// SIMATIC STEP 7 (V5.x) project hhh_v1_bisai_7_20_20_40
// CPU: CPU 412-3 H
// station: Hardware
// station: SIMATIC 400(1)
// station: P_ADR_BUS
// station: Configuration
// station: PCStation
// station: P_ADR_BUS
// program: S7 Program(1)

SYMBOL_TABLE
"OP_A_LIM"	FB 46	FB 46	// Analog value operating (limited)
"CTRL_PID"	FB 61	FB 61	// PID Control
"MEAS_MON"	FB 65	FB 65	// Meas.value monitoring block
"CONEC"	FB 88	FB 88	// Connection Function Block
"PS"	FB 89	FB 89	// Power Supply Function Block
"OB_BEGIN"	FB 100	FB 100	// CPU Function Block
"SUBNET"	FB 106	FB 106	// SUBNET Function Block
"RACK"	FB 107	FB 107	// RACK Function Block
"OB_DIAG1"	FB 118	FB 118	// OB Diagnostic Function
"CPU_RT"	FB 128	FB 128	// CPU Performance Block
"@SFC_BZL"	FB 245	FB 245	// SFC-State Logic
"@SFC_ESM"	FB 246	FB 246	// SFC-Extended State Management
"@SFC_RTS"	FB 300	FB 300	// SFC-Run-Time System V6
"SUB_R"	FC 62	FC 62	// REAL-Subtraction
"@SFC_INDCALL"	FC 250	FC 250	// SFC-Indirect-Call Function
"ADD4_P"	FC 256	FC 256	// Adder with 4 inputs
"ChkREAL"	FC 260	FC 260	// Check infinite values
"MUL4_P"	FC 262	FC 262	// Multiplier with 4 inputs
"CH_AI"	FC 275	FC 275	// Analog Input
"CH_AO"	FC 276	FC 276	// Analog Output
"PO_UPDAT"	FC 279	FC 279	// Update Process Output
"OB_END"	FC 280	FC 280	// Terminate OB Function Block
"FI1106"	IW 512	WORD	// 产品D混合物料流量
"FI1101"	IW 514	WORD	// 原料A流量
"FI1102"	IW 516	WORD	// 原料B流量
"FI1103"	IW 518	WORD	// 原料混合进料流量
"FI1104"	IW 520	WORD	// 催化剂C流量
"FI1105"	IW 522	WORD	// 反应生成液流量
"FI1107"	IW 524	WORD	//  闪蒸罐顶部循环原料A流量
"FI1201"	IW 526	WORD	// 反应器R101夹套循环上水流量
"FI1202"	IW 528	WORD	//  反应器R101夹套循环回水至预热器流量
"FI1203"	IW 530	WORD	//  反应器R101夹套循环回水至界区流量
"LI1101"	IW 532	WORD	//  混合罐V101液位
"LI1102"	IW 534	WORD	//  反应器R101液位
"LI1201"	IW 536	WORD	//  闪蒸罐V102液位
"TI1101"	IW 538	WORD	//  混合罐V101温度
"TI1102"	IW 540	WORD	//  原料混合进料出预热器E101温度
"TI1103"	IW 542	WORD	//  反应器R101温度
"TI1104"	IW 544	WORD	// 闪蒸罐V102温度
"TI1105"	IW 546	WORD	//  反应器R101夹套循环回水温度
"TI1201"	IW 548	WORD	//  反应器R101夹套循环回水出预热器温度
"aaa"	IW 550	WORD
"PI1101"	IW 552	WORD	//   混合罐压力
"PI1102"	IW 554	WORD	//  反应器压力
"PI1103"	IW 556	WORD	//  闪蒸罐压力
"xxx"	IW 558	WORD
"AI1101"	IW 564	WORD	//  产物中产品D含量
"6"	Q 0.1	BOOL
"aa"	Q 0.5	BOOL
"bb"	Q 0.6	BOOL
"cc"	Q 0.7	BOOL
"4"	Q 1.0	BOOL
"5"	Q 1.2	BOOL
"XV1101"	Q 2.1	BOOL	// 抑制剂管线阀门
"HS1105"	Q 2.2	BOOL	// D输送泵P105开关
"HS1101"	Q 2.5	BOOL	//  A进料泵P101开关
"HS1102"	Q 2.6	BOOL	//  B进料泵P102开关
"HS1103"	Q 2.7	BOOL	//  催化剂输送泵P103开关
"HS1104"	Q 3.0	BOOL	//  真空泵P104开关
"FV1106"	QW 512	WORD	// 闪蒸罐V102底部产品D管线阀门
"PV1101"	QW 514	WORD	// 闪蒸罐V102顶部循环原料A管线阀门
"FV1101"	QW 516	WORD	//  原料A管线阀门
"FV1102"	QW 518	WORD	//  原料B管线阀门
"FV1103"	QW 520	WORD	// 混合罐V101底部混合进料管线阀门
"FV1104"	QW 522	WORD	//  催化剂C管线阀门
"S1101"	QW 524	WORD	//  变频真空泵频率
"FV1105"	QW 526	WORD	//  反应器R101底部反应生成液管线阀门
"xx"	QW 528	WORD
"xxxx"	QW 530	WORD
"xxxxx"	QW 532	WORD
"FV1201"	QW 534	WORD	//  反应器R101夹套循环上水管线阀门
"FV1202"	QW 536	WORD	//  反应器R101夹套循环回水至预热器管线阀门
"FV1203"	QW 538	WORD	//  反应器R101夹套循环回水至界区管线阀门
"ALARM_8P"	SFB 35	SFB 35	// Generate Block-Related Messages with Values for 8 Signals
"NOTIFY"	SFB 36	SFB 36	// Generate Block-Related Messages without Acknowledgment Display
"RDREC"	SFB 52	SFB 52	// Read a Process Data Record
"RALRM"	SFB 54	SFB 54	// Receive Alarm Data
"BLKMOV"	SFC 20	SFC 20	// Copy Variables
END_SYMBOL_TABLE
